{attribute 'GeneratedUsingTerminal: EL6720-0000-0016'}
{attribute addProperty BoxType "EL6720-0000-0016"}
{attribute addProperty Id "EtcSlaveTerminalBaseInfoDataAT %I*InfoData_90184F0C16"}
{attribute addProperty CRC "354618671"}
{attribute addProperty Size "16"}
TYPE EL6720_15230D2F EXTENDS EtcSlaveTerminalBase :
STRUCT
	{attribute addProperty Name "InfoData"}
	InfoData : InfoData_90184F0C;
END_STRUCT
END_TYPE

(* stored: Version 1.2.0.0, ProductVersion 3.1.4024.9
   DUT EL6720_15230D2F: Id {5a33c83c-6e6c-4963-ac54-5e0ec65e4ee9} *)
